# EPICS substitutions: iocBoot/iocoh26/substitutions/canberra_3.substitutions
file "$(MCA)/mcaApp/Db/simple_mca.db"
{
pattern
{P           M       DTYP           INP              PREC  CHANS}
{oh26:med:   mca1  "asynMCA"       "@asyn(AIM1/1 0)"  3     2048}
{oh26:med:   mca2  "asynMCA"       "@asyn(AIM1/2 0)"  3     2048}
{oh26:med:   mca3  "asynMCA"       "@asyn(AIM2/1 0)"  3     2048}
{oh26:med:   mca0  "Soft Channel"  ""                 3     2048}
}

#file "$(MCA)/mcaApp/Db/icb_amp.db"
#{
#pattern
#{P			AMP		PORT}
#{oh26:med:	amp1	icbAmp1}
#}

file "$(MCA)/mcaApp/Db/icb_adc.db"
{
pattern
{P			ADC		PORT}
{oh26:med:	adc1	"icbAdc1"}
{oh26:med:	adc2	"icbAdc2"}
{oh26:med:	adc3	"icbAdc3"}
}

#file "$(MCA)/mcaApp/Db/icb_hvps.db"
#{
#pattern
#{P			HVPS	LIMIT	PORT}
#{oh26:med:	hvps1	1000	"icbHvps1"}
#}

file "$(MCA)/mcaApp/Db/icb_tca.db"
{
pattern
{P,          TCA,	PORT,		MCA}
{oh26:med:,  tca1,	"icbTca1",	mca1}
{oh26:med:,  tca2,	"icbTca2",	mca2}
{oh26:med:,  tca3,	"icbTca3",	mca3}
}
